PROGRAM MAIN
VAR
END_VAR

END_PROGRAM

(* stored: Version 1.1.0.1
   POU MAIN: Id {38a10a06-a8a5-4a8f-92f3-d56125e5d3b4}, SpecialFunc None *)
